PROGRAM ModbusRTU_EL
VAR
(*Modbus für Klemme EL6021 wird deklariert*)
	ModbusEL6021:		ModbusRtuMaster_KL6x22B;	
	modbusTimeout_EL:	TIME := T#300MS;
	isModbusBusy_EL:	BOOL;
	isModbusError_EL:	BOOL;
	modbusErrorId_EL:	MODBUS_ERRORS;
	
(*Hilfsvariablen für Modbus	

Sensor/Aktor	|	Position		|	Modbus-Adresse
________________|___________________|____________________
EV				|	3				|	2
EV_rev			|	3				|	3	
*)
	//modbusData_EV: 	ARRAY[1..10] OF INT;		//hier werden die Daten vom EV gespeichert
	EV_Adresse : BYTE := 2;				//ModbusAdresse vom Expansionsventil	
	EV_rev_Adresse : BYTE := 3;			//ModbusAdresse vom Abtau-Expansionsventil
	state: 			INT := 0;
	counter: 		INT := 1;
	
	AbfrageRegs: ARRAY [1..10] OF WORD := [0,1,4,5,6,9,16,20,131,134]; 	//Modbus-Register-Adressen. Das sind alle Werte die vom EV abgefragt werden
	AbfrageCoils: ARRAY [1..4] OF WORD := [49,50,51,52];					//Modbus-Coil-Adressen.
	
(*Variablen für Error- und Successzähler der Modbus-Komunikation *)
	FtrigBusy:			F_TRIG;
	LastErrorstate: 	INT;
	LastModbusError: 	ST_ModbusErrorDiagnostics;
	CounterError: 		DINT;
	CounterSuccess: 	DINT;

	TestMSS: ARRAY [0..10] OF DWORD;
END_VAR


CASE state OF

0: (*Initialisierung von Modbus*)
	
		ModbusEL6021.ReadInputRegs(Execute:= FALSE);
		ModbusEL6021.ReadCoils(Execute:= FALSE);
		ModbusEL6021.WriteSingleRegister(Execute:= FALSE);

		state :=1;
		
1: (*Liest Register von EV aus*)
 	
		ModbusEL6021.ReadInputRegs(
		UnitID:= EV_Adresse,
 		Quantity:= 1,								
 		MBAddr:= AbfrageRegs[counter],								
 		cbLength:= SIZEOF(EV.modbusData[counter]),//EV.modbusData[counter]),		
 		pMemoryAddr:= ADR(EV.modbusData[counter]),//EV.modbusData[counter]),		//Daten werden in für EV DATA-ARRAY geschrieben
  		Execute:= TRUE,
  		Timeout:= modbusTimeout_EL,
  		Busy => isModbusBusy_EL,
  		Error => isModbusError_EL,
  		ErrorId => modbusErrorId_EL
  		(*cbRead parameter)*));

		IF NOT isModbusBusy_EL THEN
				ModbusEL6021.ReadInputRegs(Execute:= FALSE);
			IF MODBUS.myModbus.Error THEN
				state := 0;
				ELSE
				counter := counter + 1;	
					IF counter > 10 THEN		//alle deklarierten Modbus-Register werden ausgelesen
					counter := 1;
					state:= 2;
					END_IF
			END_IF
		END_IF
		


	
2: (*Liest Coils von EV aus*)
		ModbusEL6021.ReadCoils(
		UnitID:= EV_Adresse,
 		Quantity:= 1,								
 		MBAddr:= AbfrageCoils[counter],								
 		cbLength:= SIZEOF(EV.modbusDataCoils[counter]),		
 		pMemoryAddr:= ADR(EV.modbusDataCoils[counter]),		//Daten werden in für EV DATA-ARRAY geschrieben
  		Execute:= TRUE,
  		Timeout:= modbusTimeout_EL,
  		Busy => isModbusBusy_EL,
  		Error => isModbusError_EL,
  		ErrorId => modbusErrorId_EL
  		(*cbRead parameter)*));
		
		IF NOT isModbusBusy_EL THEN
				ModbusEL6021.ReadCoils(Execute:= FALSE);
			IF ModbusEL6021.Error THEN
				state := 0;
			ELSE
				counter:= counter+1;
				IF counter > 4 THEN		//alle deklarierten Modbus-Register werden ausgelesen
					counter := 1;
					state:= 3;
				END_IF
			END_IF
		END_IF
		
3: (*Schreibt Akt_Kühlleistung Coil auf die Expansionsventile*)
IF EV.SetKuhlleistung THEN 	
	ModbusEL6021.WriteSingleRegister(
		UnitID:= EV_Adresse,
 		Quantity:= 1,								
 		MBAddr:= 134,								
 		cbLength:= SIZEOF(EV.SollKuhlleistung),		
 		pMemoryAddr:= ADR(EV.SollKuhlleistung),		//Daten werden in für EV DATA-ARRAY geschrieben
  		Execute:= TRUE,
  		Timeout:= modbusTimeout_EL,
  		Busy => isModbusBusy_EL,
  		Error => isModbusError_EL,
  		ErrorId => modbusErrorId_EL
  		(*cbRead parameter)*));

		IF NOT isModbusBusy_EL THEN
				ModbusEL6021.WriteSingleRegister(Execute:= FALSE);
				EV.SetKuhlleistung := FALSE;
			IF ModbusEL6021.Error THEN
				state := 0;
			ELSE
				state:= 4;
			END_IF
		END_IF
	ELSE 
		state:= 4;
END_IF
	
4: (*Liest Register von EV_rev aus*)
 	
		ModbusEL6021.ReadInputRegs(
		UnitID:= EV_rev_Adresse,
 		Quantity:= 1,								
 		MBAddr:= AbfrageRegs[counter],								
 		cbLength:= SIZEOF(EV_rev.modbusData[counter]),//EV.modbusData[counter]),		
 		pMemoryAddr:= ADR(EV_rev.modbusData[counter]),//EV.modbusData[counter]),		//Daten werden in für EV DATA-ARRAY geschrieben
  		Execute:= TRUE,
  		Timeout:= modbusTimeout_EL,
  		Busy => isModbusBusy_EL,
  		Error => isModbusError_EL,
  		ErrorId => modbusErrorId_EL
  		(*cbRead parameter)*));

		IF NOT isModbusBusy_EL THEN
				ModbusEL6021.ReadInputRegs(Execute:= FALSE);
			IF MODBUS.myModbus.Error THEN
				state := 0;
				ELSE
				counter := counter + 1;	
					IF counter > 10 THEN		//alle deklarierten Modbus-Register werden ausgelesen
					counter := 1;
					state:= 5;
					END_IF
			END_IF
		END_IF
		


	
5: (*Liest Coils von EV_rev aus*)
		

		ModbusEL6021.ReadCoils(
		UnitID:= EV_rev_Adresse,
 		Quantity:= 1,								
 		MBAddr:= AbfrageCoils[counter],								
 		cbLength:= SIZEOF(EV_rev.modbusDataCoils[counter]),		
 		pMemoryAddr:= ADR(EV_rev.modbusDataCoils[counter]),		//Daten werden in für EV DATA-ARRAY geschrieben
  		Execute:= TRUE,
  		Timeout:= modbusTimeout_EL,
  		Busy => isModbusBusy_EL,
  		Error => isModbusError_EL,
  		ErrorId => modbusErrorId_EL
  		(*cbRead parameter)*));

		IF NOT isModbusBusy_EL THEN
				ModbusEL6021.ReadCoils(Execute:= FALSE);
			IF ModbusEL6021.Error THEN
				state := 0;
			ELSE
				counter:= counter+1;
				IF counter > 4 THEN		//alle deklarierten Modbus-Register werden ausgelesen
					counter := 1;
					state:= 6;
				END_IF
			END_IF

		END_IF

6: (*Schreibt Akt_Kühlleistung Coil auf die Expansionsventile*)

IF EV_rev.SetKuhlleistung THEN 	
	ModbusEL6021.WriteSingleRegister(
		UnitID:= EV_rev_Adresse,
 		Quantity:= 1,								
 		MBAddr:= 134,								
 		cbLength:= SIZEOF(EV_rev.SollKuhlleistung),		
 		pMemoryAddr:= ADR(EV_rev.SollKuhlleistung),		//Daten werden in für EV DATA-ARRAY geschrieben
  		Execute:= TRUE,
  		Timeout:= modbusTimeout_EL,
  		Busy => isModbusBusy_EL,
  		Error => isModbusError_EL,
  		ErrorId => modbusErrorId_EL
  		(*cbRead parameter)*));

		IF NOT isModbusBusy_EL THEN
				ModbusEL6021.WriteSingleRegister(Execute:= FALSE);
				EV_rev.SetKuhlleistung := FALSE;
			IF ModbusEL6021.Error THEN
				state := 0;
			ELSE
				state:= 0;
			END_IF
		END_IF
	ELSE 
		state:= 0;
END_IF	
END_CASE

FtrigBusy(CLK:=ModbusEL6021.BUSY );
(*zählt fehlgeschlagene und erfolgreiche Komunikationsschritte*)
IF FtrigBusy.Q THEN
	IF ModbusEL6021.Error THEN
		LastModbusError := ModbusEL6021.ErrorDiagnostics;
		LastErrorstate := state;
		CounterError := CounterError + 1;
	ELSE
		CounterSuccess := CounterSuccess + 1;
	END_IF
END_IF

END_PROGRAM

(* stored: Version 1.1.0.1, ProductVersion 3.1.4019.2
   POU ModbusRTU_EL: Id {98159f27-7da7-4f3a-9d45-35bf24bd6264}, SpecialFunc None *)
